// TwinCAT 3 PLC project MemRingBufferExample
// ProgramVersion: 3.1.0.8
// libraries:
//   Tc2_Standard, * (Beckhoff Automation GmbH)
//   Tc2_System, * (Beckhoff Automation GmbH)
//   Tc2_Utilities, * (Beckhoff Automation GmbH)
//   Tc3_Interfaces, * (Beckhoff Automation GmbH)
//   Tc3_Module, * (Beckhoff Automation GmbH)
// project tree:
//   DUTs/ ST_DataSetEntry.TcDUT (not stored)
//   GVLs/ GVL.TcGVL
//   POUs/ FB_DataSetFifo.TcPOU, MAIN.TcPOU
//   / Standard.TcTTO
// (motion and I/O tree: see PLC project untitled1)
// real-time tasks:
//   TASK PlcTask: cycle T#10ms, priority 20, ADS port 350
//   TASK PlcTask1: cycle T#10ms, priority 21, ADS port 351

CONFIGURATION MemRingBufferExample
    RESOURCE PLC ON TwinCAT3
        TASK Standard(INTERVAL := T#10ms, PRIORITY := 20);
        PROGRAM MAIN WITH Standard : MAIN;
    END_RESOURCE
END_CONFIGURATION

// ---- GVLs/GVL.TcGVL
VAR_GLOBAL CONSTANT
	MAX_BUFFER_SIZE : UDINT := 1000;
END_VAR

// ---- POUs/MAIN.TcPOU
PROGRAM MAIN
VAR
	fbFifo 		: FB_DataSetFifo := ( bOverwrite := TRUE );
	newEntry	: ST_DataSetEntry;
	oldEntry	: ST_DataSetEntry;
	bSuccess	: BOOL;
	nCount		: UDINT;
	nLoad		: UDINT;

	bReset 		: BOOL := TRUE;
	bAdd 		: BOOL := TRUE;
	bGet		: BOOL := TRUE;
	bRemove		: BOOL := TRUE;
END_VAR

IF bReset THEN
	bReset := FALSE;
	(* reset fifo (clear all entries) *)
	fbFifo.A_Reset(	in := newEntry, bOk=>bSuccess, nCount=> nCount, nLoad => nLoad );
END_IF

IF bAdd THEN
	bAdd := FALSE;

	(* create new or modify data set entry *)
	newEntry.bFlag := NOT newEntry.bFlag;
	newEntry.nValue := newEntry.nValue + 1;
	newEntry.sMsg := BYTE_TO_STRING(newEntry.nValue);

	(* add new entry to the fifo *)
	fbFifo.A_Add(	in := newEntry, bOk=>bSuccess, nCount=> nCount, nLoad => nLoad );
END_IF

IF bGet THEN
	bGet := FALSE;
	(* get (but not delete) oldest entry *)
	fbFifo.A_Get( out => oldEntry, bOk => bSuccess, nCount => nCount, nLoad => nLoad );
END_IF

IF bRemove THEN
	bRemove:= FALSE;
	(* remove oldest entry *)
	fbFifo.A_Remove( out => oldEntry, bOk => bSuccess, nCount => nCount, nLoad => nLoad );
END_IF

END_PROGRAM

// ---- POUs/FB_DataSetFifo.TcPOU
FUNCTION_BLOCK FB_DataSetFifo
VAR_INPUT
	bOverwrite	: BOOL;
	in 			: ST_DataSetEntry;
END_VAR
VAR_OUTPUT
	bOk			: BOOL;
	nCount		: UDINT;
	nLoad		: UDINT;
	out			: ST_DataSetEntry;
END_VAR
VAR
	arrBuffer 	: ARRAY[0..MAX_BUFFER_SIZE] OF BYTE; (* Buffer memory used by FB_MemRingBuffer function block *)
	fbBuffer	: FB_MemRingBuffer;
END_VAR

;

ACTION A_Reset:
MEMSET( ADR( arrBuffer ), 0, SIZEOF( arrBuffer ) ); (* reset (optional) internal buffer *)

fbBuffer.A_Reset( 	bOk=> bOk,
					nCount => nCount );

nLoad := (fbBuffer.cbSize * 100) / MAX_BUFFER_SIZE;
END_ACTION

ACTION A_Remove:
fbBuffer.A_RemoveHead( 	pRead:= ADR( out ),
						cbRead:= SIZEOF( out ),
						pBuffer:= ADR( arrBuffer ),
						cbBuffer:= SIZEOF( arrBuffer ),
						bOk=> bOk,
						nCount => nCount );

nLoad := (fbBuffer.cbSize * 100) / MAX_BUFFER_SIZE;
END_ACTION

ACTION A_Get:
fbBuffer.A_GetHead( pRead:= ADR( out ),
					cbRead:= SIZEOF( out ),
					pBuffer:= ADR( arrBuffer ),
					cbBuffer:= SIZEOF( arrBuffer ),
					bOk=> bOk,
					nCount => nCount );

nLoad := (fbBuffer.cbSize * 100) / MAX_BUFFER_SIZE;
END_ACTION

ACTION A_Add:
fbBuffer.A_AddTail( pWrite:= ADR( in ),
					cbWrite:= SIZEOF( in ),
					pBuffer:= ADR( arrBuffer ),
					cbBuffer:= SIZEOF( arrBuffer ),
					bOk=> bOk,
					nCount => nCount );


IF NOT bOk THEN (* overflow ? *)
	IF bOverwrite THEN
		fbBuffer.A_RemoveHead(); (* remove one oldest entry *)

		fbBuffer.A_AddTail( bOk => bOk, nCount => nCount );
	END_IF
END_IF



nLoad := (fbBuffer.cbSize * 100) / MAX_BUFFER_SIZE;
END_ACTION

END_FUNCTION_BLOCK
